(* PLC project io_engine_1d2s, Dassault Systèmes ControlBuild 2024x *)
(* stored: creationDateTime 2023-10-03T11:12:46-01:00 *)

PROGRAM panel
  VAR_OUTPUT
    highSpeedPB : BOOL := false;
    lowSpeedPB : BOOL := false;
    stopPB : BOOL := false;
  END_VAR

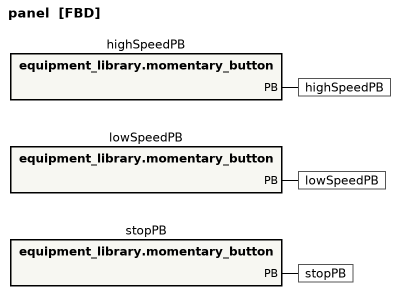
(* FBD diagram, written out as Structured Text *)
highSpeedPB();
highSpeedPB := highSpeedPB.PB;
lowSpeedPB();
lowSpeedPB := lowSpeedPB.PB;
stopPB();
stopPB := stopPB.PB;
END_PROGRAM

(* Integrated object C/C+OP of a motor with two speed and one direction *)
PROGRAM io_library.io_engine_1d2s
  VAR_INPUT
    autoMode : BOOL := false;
    manualMode : BOOL := false;
  END_VAR
  VAR_INPUT
    autoHSCmd : BOOL := false;
    autoLSCmd : BOOL := false;
  END_VAR
  VAR_INPUT
    acknowledgePB : BOOL := false;
  END_VAR
  VAR_OUTPUT
    speedVal : REAL := 0.0;
    speedPercent : REAL := 0.0;
  END_VAR
  VAR_OUTPUT
    generalFault : BOOL := false;
  END_VAR

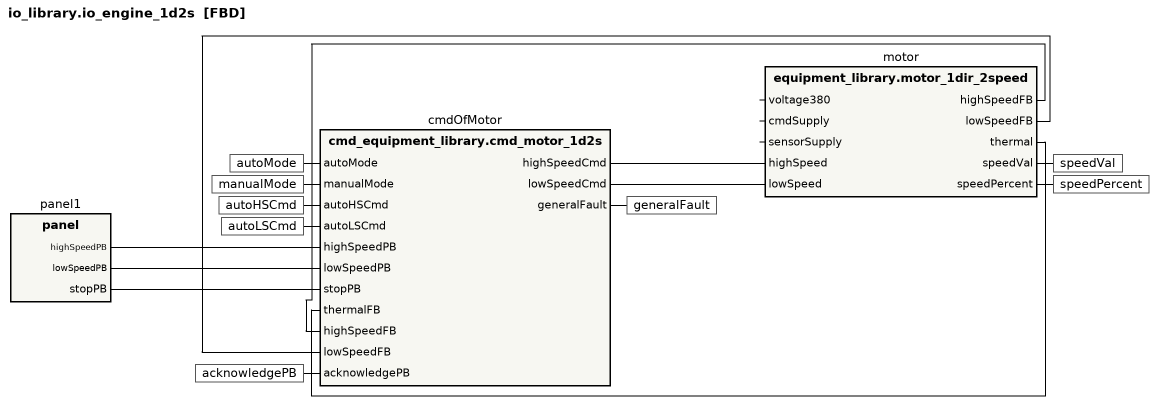
(* FBD diagram, written out as Structured Text *)
panel1();
motor(highSpeed := cmdOfMotor.highSpeedCmd, lowSpeed := cmdOfMotor.lowSpeedCmd);
cmdOfMotor(autoMode := autoMode, manualMode := manualMode, autoHSCmd := autoHSCmd, autoLSCmd := autoLSCmd, highSpeedPB := panel1.highSpeedPB, lowSpeedPB := panel1.lowSpeedPB, stopPB := panel1.stopPB, thermalFB := motor.thermal, highSpeedFB := motor.highSpeedFB, lowSpeedFB := motor.lowSpeedFB, acknowledgePB := acknowledgePB);
generalFault := cmdOfMotor.generalFault;
speedVal := motor.speedVal;
speedPercent := motor.speedPercent;
END_PROGRAM
